// TwinCAT 3 PLC project Untitled1
// ProgramVersion: 3.1.4022.7
// libraries:
//   Tc2_Standard, * (Beckhoff Automation GmbH)
//   Tc2_System, * (Beckhoff Automation GmbH)
//   Tc3_Module, * (Beckhoff Automation GmbH)
// project tree:
//   CIF/ alg_a_DledQ1.TcPOU, alg_a_DledQ2.TcPOU, alg_a_Dresetled.TcPOU, alg_a_Dstartled.TcPOU, alg_a_ejectpulse.TcPOU, alg_a_gripperclose.TcPOU, alg_a_handlingready.TcPOU, alg_a_HledQ1.TcPOU, alg_a_HledQ2.TcPOU, alg_a_Hresetled.TcPOU, alg_a_Hstartled.TcPOU, alg_a_pusher1.TcPOU, alg_a_pusher2.TcPOU, alg_a_pusher3.TcPOU, alg_a_transfer2droppos.TcPOU, alg_a_transfer2pickpos.TcPOU, alg_a_vacuum.TcPOU, alg_a_x2distributing.TcPOU, alg_a_x2testing.TcPOU, alg_a_zdown.TcPOU, alg_M_example_controller_a_Dstartled.TcPOU, alg_M_example_controller_godown.TcPOU, alg_s_Dinitialized.TcPOU, alg_s_Hinitialized.TcPOU, derivcvar_M_HardwareMap_t.TcPOU, enum_E.TcDUT, INPUTS.TcGVL, MAIN.TcPOU, makeArray0.TcPOU, normProjIdx.TcPOU, projArray0.TcPOU, STATE.TcDUT, TIMERS.TcGVL
//   / PlcTask.TcTTO
//   UNITY/ ACTUATOR.TcPOU (not stored), GVLS.TcGVL (not stored), INDICATORLIGHT.TcPOU (not stored), UNITY.TcPOU
// real-time tasks:
//   TASK PlcTask: cycle T#10ms, priority 20, ADS port 350

CONFIGURATION Untitled1
    RESOURCE PLC ON TwinCAT3
        TASK PlcTask(INTERVAL := T#10ms, PRIORITY := 20);
        PROGRAM MAIN WITH PlcTask : MAIN;
        PROGRAM UNITY WITH PlcTask : UNITY;
    END_RESOURCE
END_CONFIGURATION

// ---- CIF/enum_E.TcDUT
TYPE enum_E :
(
	elit_gopickup,
	elit_init0,
	elit_init1,
	elit_init2,
	elit_init3,
	elit_init4,
	elit_init5,
	elit_init6,
	elit_init7,
	elit_init8,
	elit_init9,
	elit_init_error,
	elit_init_ok,
	elit_init_sensor_check,
	elit_initialized,
	elit_running,
	elit_starting,
	elit_wait_init,
	elit_wait_start
);
END_TYPE

// ---- CIF/STATE.TcDUT
TYPE STATE :
STRUCT
	curTime: LREAL;
	dvar_M_example_controller_a_x2distributing AT %Q*: BOOL;
	dvar_M_example_controller_a_zdown AT %Q*: BOOL;
	dvar_M_example_controller_count AT %Q*: DINT;
	dvar_M_example_controller AT %Q*: enum_E;
	dvar_M_HardwareMap_out_a_Dstartled AT %Q*: BOOL;
	dvar_M_HardwareMap_out_a_Dresetled AT %Q*: BOOL;
	dvar_M_HardwareMap_out_a_DledQ1 AT %Q*: BOOL;
	dvar_M_HardwareMap_out_a_DledQ2 AT %Q*: BOOL;
	dvar_M_HardwareMap_out_a_Dout4 AT %Q*: BOOL;
	dvar_M_HardwareMap_out_a_Dout5 AT %Q*: BOOL;
	dvar_M_HardwareMap_out_a_Dout6 AT %Q*: BOOL;
	dvar_M_HardwareMap_out_a_Dout7 AT %Q*: BOOL;
	dvar_M_HardwareMap_out_a_pusher1 AT %Q*: BOOL;
	dvar_M_HardwareMap_out_a_pusher2 AT %Q*: BOOL;
	dvar_M_HardwareMap_out_a_pusher3 AT %Q*: BOOL;
	dvar_M_HardwareMap_out_a_Hstartled AT %Q*: BOOL;
	dvar_M_HardwareMap_out_a_Hresetled AT %Q*: BOOL;
	dvar_M_HardwareMap_out_a_HledQ1 AT %Q*: BOOL;
	dvar_M_HardwareMap_out_a_HledQ2 AT %Q*: BOOL;
	dvar_M_HardwareMap_out_a_Hout4 AT %Q*: BOOL;
	dvar_M_HardwareMap_out_a_Hout5 AT %Q*: BOOL;
	dvar_M_HardwareMap_out_a_Hout6 AT %Q*: BOOL;
	dvar_M_HardwareMap_out_a_Hout7 AT %Q*: BOOL;
	dvar_M_HardwareMap_out_a_x2distributing AT %Q*: BOOL;
	dvar_M_HardwareMap_out_a_x2testing AT %Q*: BOOL;
	dvar_M_HardwareMap_out_a_zdown AT %Q*: BOOL;
	dvar_M_HardwareMap_out_a_gripperclose AT %Q*: BOOL;
	dvar_M_HardwareMap_out_a_transfer2pickpos AT %Q*: BOOL;
	dvar_M_HardwareMap_out_a_transfer2droppos AT %Q*: BOOL;
	dvar_M_HardwareMap_out_a_vacuum AT %Q*: BOOL;
	dvar_M_HardwareMap_out_a_ejectpulse AT %Q*: BOOL;
	dvar_M_HardwareMap_out_a_handlingready AT %Q*: BOOL;
	dvar_M_HardwareMap_init_err_sen_idx AT %Q*: DINT;
	dvar_M_HardwareMap_init_err_led_idx AT %Q*: DINT;
	cvar_M_HardwareMap_t AT %Q*: LREAL;
	dvar_M_HardwareMap AT %Q*: enum_E;
END_STRUCT
END_TYPE

// ---- CIF/INPUTS.TcGVL
VAR_GLOBAL
	ivar_s_Dstartbutton AT %I*: BOOL;
	ivar_s_Dstopbutton AT %I*: BOOL;
	ivar_s_Dresetbutton AT %I*: BOOL;
	ivar_s_Dautoswitch AT %I*: BOOL;
	ivar_s_pusher1_in AT %I*: BOOL;
	ivar_s_pusher1_out AT %I*: BOOL;
	ivar_s_stack1filled AT %I*: BOOL;
	ivar_s_product1 AT %I*: BOOL;
	ivar_s_pusher2_in AT %I*: BOOL;
	ivar_s_pusher2_out AT %I*: BOOL;
	ivar_s_stack2filled AT %I*: BOOL;
	ivar_s_product2 AT %I*: BOOL;
	ivar_s_pusher3_in AT %I*: BOOL;
	ivar_s_pusher3_out AT %I*: BOOL;
	ivar_s_stack3filled AT %I*: BOOL;
	ivar_s_product3 AT %I*: BOOL;
	ivar_s_handlingbusy AT %I*: BOOL;
	ivar_s_Hstartbutton AT %I*: BOOL;
	ivar_s_Hstopbutton AT %I*: BOOL;
	ivar_s_Hresetbutton AT %I*: BOOL;
	ivar_s_Hautoswitch AT %I*: BOOL;
	ivar_s_xpos_at1 AT %I*: BOOL;
	ivar_s_xpos_at2 AT %I*: BOOL;
	ivar_s_xpos_at3 AT %I*: BOOL;
	ivar_s_xpos_atdrop AT %I*: BOOL;
	ivar_s_zpos_atup AT %I*: BOOL;
	ivar_s_zpos_atdown AT %I*: BOOL;
	ivar_s_gripper AT %I*: BOOL;
	ivar_s_transfer_atpickup AT %I*: BOOL;
	ivar_s_transfer_atdrop AT %I*: BOOL;
	ivar_s_transfer_athalfway AT %I*: BOOL;
	ivar_s_vacuum AT %I*: BOOL;
	ivar_s_product4 AT %I*: BOOL;
	ivar_s_testingbusy AT %I*: BOOL;
	ivar_s_Din4 AT %I*: BOOL;
	ivar_s_Din5 AT %I*: BOOL;
	ivar_s_Din6 AT %I*: BOOL;
	ivar_s_Din7 AT %I*: BOOL;
	ivar_s_Hin4 AT %I*: BOOL;
	ivar_s_Hin5 AT %I*: BOOL;
	ivar_s_Hin6 AT %I*: BOOL;
	ivar_s_Hin7 AT %I*: BOOL;
	ivar_a_Dout4 AT %I*: BOOL;
	ivar_a_Dout5 AT %I*: BOOL;
	ivar_a_Dout6 AT %I*: BOOL;
	ivar_a_Dout7 AT %I*: BOOL;
	ivar_a_Hout4 AT %I*: BOOL;
	ivar_a_Hout5 AT %I*: BOOL;
	ivar_a_Hout6 AT %I*: BOOL;
	ivar_a_Hout7 AT %I*: BOOL;
END_VAR

// ---- CIF/TIMERS.TcGVL
VAR_GLOBAL
	timer0: TON;
	timer1: TON;
	curTimer: INT := 0;
END_VAR

// ---- CIF/MAIN.TcPOU
PROGRAM MAIN
VAR_OUTPUT
	timerValue0: TIME;
	timerValue1: TIME;
END_VAR
VAR
	cnt: LINT;
	first: BOOL := TRUE;
	curTimerValue: TIME;
	state0: STATE;
	curTime: LREAL;
	loopsKilled: LINT;
END_VAR
VAR_TEMP
	lastTimerValue: TIME;
	curDeltaTime: TIME;
	curDeltaSecs: LREAL;
	state1: STATE;
	progress: BOOL;
	loopCount: INT;
	b1: BOOL;
	b2: BOOL;
END_VAR


// Handle 'time' and cycle time.
cnt := cnt + 1;

timer0(IN := curTimer = 0, PT := T#1D);
timer1(IN := curTimer = 1, PT := T#1D);
timerValue0 := timer0.ET;
timerValue1 := timer1.ET;

lastTimerValue := curTimerValue;
IF curTimer = 0 THEN
    curTimerValue := timerValue0;
ELSE
    curTimerValue := timerValue1;
END_IF;
curDeltaTime := curTimerValue - lastTimerValue;
curDeltaSecs := TIME_TO_LREAL(curDeltaTime) / 1000;
curTime := curTime + curDeltaSecs;

IF cnt MOD 10 = 0 THEN
    curTimer := 1 - curTimer;
    curTimerValue := T#0S;
    timer0(IN := curTimer = 0, PT := T#1D);
    timer1(IN := curTimer = 1, PT := T#1D);
    timerValue0 := timer0.ET;
    timerValue1 := timer1.ET;
END_IF;

IF first THEN
    first := FALSE;

    // Initialize state variables for initial state.
    state0.dvar_M_example_controller_a_x2distributing := FALSE;
    state0.dvar_M_example_controller_a_zdown := FALSE;
    state0.dvar_M_example_controller_a_gripperclose := FALSE;
    state0.dvar_M_example_controller_a_x2testing := FALSE;
    state0.dvar_M_example_controller_i := 0;
    state0.cvar_M_example_controller_t := 0.0;
    state0.dvar_M_example_controller := elit_init2;
    state0.dvar_M_HardwareMap_out_a_Dstartled := FALSE;
    state0.dvar_M_HardwareMap_out_a_Dresetled := FALSE;
    state0.dvar_M_HardwareMap_out_a_DledQ1 := TRUE;
    state0.dvar_M_HardwareMap_out_a_DledQ2 := TRUE;
    state0.dvar_M_HardwareMap_out_a_Dout4 := FALSE;
    state0.dvar_M_HardwareMap_out_a_Dout5 := FALSE;
    state0.dvar_M_HardwareMap_out_a_Dout6 := FALSE;
    state0.dvar_M_HardwareMap_out_a_Dout7 := FALSE;
    state0.dvar_M_HardwareMap_out_a_pusher1 := FALSE;
    state0.dvar_M_HardwareMap_out_a_pusher2 := FALSE;
    state0.dvar_M_HardwareMap_out_a_pusher3 := FALSE;
    state0.dvar_M_HardwareMap_out_a_Hstartled := FALSE;
    state0.dvar_M_HardwareMap_out_a_Hresetled := FALSE;
    state0.dvar_M_HardwareMap_out_a_HledQ1 := TRUE;
    state0.dvar_M_HardwareMap_out_a_HledQ2 := TRUE;
    state0.dvar_M_HardwareMap_out_a_Hout4 := FALSE;
    state0.dvar_M_HardwareMap_out_a_Hout5 := FALSE;
    state0.dvar_M_HardwareMap_out_a_Hout6 := FALSE;
    state0.dvar_M_HardwareMap_out_a_Hout7 := FALSE;
    state0.dvar_M_HardwareMap_out_a_x2distributing := TRUE;
    state0.dvar_M_HardwareMap_out_a_x2testing := TRUE;
    state0.dvar_M_HardwareMap_out_a_zdown := FALSE;
    state0.dvar_M_HardwareMap_out_a_gripperclose := FALSE;
    state0.dvar_M_HardwareMap_out_a_transfer2pickpos := FALSE;
    state0.dvar_M_HardwareMap_out_a_transfer2droppos := FALSE;
    state0.dvar_M_HardwareMap_out_a_vacuum := FALSE;
    state0.dvar_M_HardwareMap_out_a_ejectpulse := FALSE;
    state0.dvar_M_HardwareMap_out_a_handlingready := FALSE;
    state0.dvar_M_HardwareMap_init_err_sen_idx := -1;
    state0.dvar_M_HardwareMap_init_err_led_idx := 0;
    state0.cvar_M_HardwareMap_t := 0.0;
    state0.dvar_M_HardwareMap := elit_init0;
    state0.dvar_M_inventory1_a_pusher1 := FALSE;
    state0.dvar_M_inventory1 := elit_init2;
    state0.dvar_M_inventory2_a_pusher2 := FALSE;
    state0.dvar_M_inventory2 := elit_init2;
    state0.dvar_M_inventory3_a_pusher3 := FALSE;
    state0.dvar_M_inventory3 := elit_init2;
    state0.dvar_M_vacuum_a_transfer2pickpos := FALSE;
    state0.dvar_M_vacuum_a_transfer2droppos := FALSE;
    state0.dvar_M_vacuum_a_vacuum := FALSE;
    state0.dvar_M_vacuum_a_ejectpulse := FALSE;
    state0.dvar_M_vacuum := elit_init2;
ELSE
    // Update continuous variables for time delay.
    state1.cvar_M_example_controller_t := state0.cvar_M_example_controller_t + curDeltaSecs * derivcvar_M_example_controller_t(state0);
    state1.cvar_M_HardwareMap_t := state0.cvar_M_HardwareMap_t + curDeltaSecs * derivcvar_M_HardwareMap_t(state0);

    state0.curTime := curTime;
    state0.cvar_M_example_controller_t := state1.cvar_M_example_controller_t;
    state0.cvar_M_HardwareMap_t := state1.cvar_M_HardwareMap_t;
END_IF;

// Event loop.
WHILE TRUE DO
    progress := FALSE;

    // Event "tau".
    IF NOT progress THEN
        b1 := (state0.dvar_M_example_controller) = (elit_init2);
        b1 := b1 AND (alg_s_Dinitialized(state0));
        IF b1 THEN
            progress := TRUE;
            state1 := state0;

            state1.dvar_M_example_controller := elit_wait_start;

            state0 := state1;
        END_IF;
    END_IF;

    // Event "tau".
    IF NOT progress THEN
        b1 := (state0.dvar_M_example_controller) = (elit_wait_start);
        b1 := b1 AND (ivar_s_Dstartbutton);
        IF b1 THEN
            progress := TRUE;
            state1 := state0;

            state1.dvar_M_example_controller := elit_droppoint;

            state0 := state1;
        END_IF;
    END_IF;

    // Event "tau".
    IF NOT progress THEN
        b1 := (state0.dvar_M_example_controller) = (elit_droppoint);
        b1 := b1 AND (ivar_s_gripper);
        b1 := b1 AND (ivar_s_xpos_atdrop);
        b1 := b1 AND (ivar_s_zpos_atup);
        IF b1 THEN
            progress := TRUE;
            state1 := state0;

            state1.dvar_M_example_controller_a_x2distributing := TRUE;
            state1.dvar_M_example_controller_a_x2testing := TRUE;
            state1.dvar_M_example_controller := elit_down;

            state0 := state1;
        END_IF;
    END_IF;

    // Event "tau".
    IF NOT progress THEN
        b1 := (state0.dvar_M_example_controller) = (elit_droppoint);
        b1 := b1 AND (NOT(ivar_s_gripper));
        b1 := b1 AND (ivar_s_xpos_atdrop);
        IF b1 THEN
            progress := TRUE;
            state1 := state0;

            state1.dvar_M_example_controller_a_x2distributing := TRUE;
            state1.dvar_M_example_controller_a_x2testing := FALSE;
            state1.dvar_M_example_controller := elit_movetopickup;

            state0 := state1;
        END_IF;
    END_IF;

    // Event "tau".
    IF NOT progress THEN
        b1 := (state0.dvar_M_example_controller) = (elit_movetopickup);
        b1 := b1 AND (projArray1(alg_M_example_controller_atpos(state0), projArray0(makeArray0(0, 1, 0, 2), state0.dvar_M_example_controller_i)));
        b1 := b1 AND ((state0.dvar_M_example_controller_i) < (3));
        IF b1 THEN
            progress := TRUE;
            state1 := state0;

            state1.dvar_M_example_controller_i := (state0.dvar_M_example_controller_i) + (1);
            state1.dvar_M_example_controller_a_x2distributing := TRUE;
            state1.dvar_M_example_controller_a_x2testing := TRUE;
            state1.dvar_M_example_controller := elit_down;

            state0 := state1;
        END_IF;
    END_IF;

    // Event "tau".
    IF NOT progress THEN
        b1 := (state0.dvar_M_example_controller) = (elit_movetopickup);
        b1 := b1 AND (projArray1(alg_M_example_controller_atpos(state0), projArray0(makeArray0(0, 1, 0, 2), state0.dvar_M_example_controller_i)));
        b1 := b1 AND ((state0.dvar_M_example_controller_i) >= (3));
        IF b1 THEN
            progress := TRUE;
            state1 := state0;

            state1.dvar_M_example_controller_i := 0;
            state1.dvar_M_example_controller_a_x2distributing := TRUE;
            state1.dvar_M_example_controller_a_x2testing := TRUE;
            state1.dvar_M_example_controller := elit_down;

            state0 := state1;
        END_IF;
    END_IF;

    // Event "tau".
    IF NOT progress THEN
        IF (state0.dvar_M_example_controller) = (elit_down) THEN
            progress := TRUE;
            state1 := state0;

            state1.dvar_M_example_controller_a_zdown := TRUE;
            state1.dvar_M_example_controller := elit_gopickup;

            state0 := state1;
        END_IF;
    END_IF;

    // Event "tau".
    IF NOT progress THEN
        b1 := (state0.dvar_M_example_controller) = (elit_gopickup);
        b1 := b1 AND (ivar_s_zpos_atdown);
        b1 := b1 AND (ivar_s_gripper);
        b1 := b1 AND (NOT(ivar_s_xpos_atdrop));
        IF b1 THEN
            progress := TRUE;
            state1 := state0;

            state1.dvar_M_example_controller_a_gripperclose := TRUE;
            state1.dvar_M_example_controller_a_zdown := FALSE;
            state1.dvar_M_example_controller := elit_goback;

            state0 := state1;
        END_IF;
    END_IF;

    // Event "tau".
    IF NOT progress THEN
        b1 := (state0.dvar_M_example_controller) = (elit_gopickup);
        b1 := b1 AND (ivar_s_zpos_atdown);
        b1 := b1 AND (ivar_s_gripper);
        b1 := b1 AND (ivar_s_xpos_atdrop);
        IF b1 THEN
            progress := TRUE;
            state1 := state0;

            state1.dvar_M_example_controller_a_gripperclose := FALSE;
            state1.dvar_M_example_controller_a_zdown := FALSE;
            state1.dvar_M_example_controller := elit_droppoint;

            state0 := state1;
        END_IF;
    END_IF;

    // Event "tau".
    IF NOT progress THEN
        b1 := (state0.dvar_M_example_controller) = (elit_gopickup);
        b1 := b1 AND (ivar_s_zpos_atdown);
        b1 := b1 AND (NOT(ivar_s_gripper));
        b1 := b1 AND (NOT(ivar_s_xpos_atdrop));
        IF b1 THEN
            progress := TRUE;
            state1 := state0;

            state1.dvar_M_example_controller_a_zdown := FALSE;
            state1.dvar_M_example_controller_a_x2distributing := FALSE;
            state1.dvar_M_example_controller_a_x2testing := TRUE;
            state1.dvar_M_example_controller := elit_finished;

            state0 := state1;
        END_IF;
    END_IF;

    // Event "tau".
    IF NOT progress THEN
        b1 := (state0.dvar_M_example_controller) = (elit_goback);
        b1 := b1 AND (ivar_s_zpos_atup);
        b1 := b1 AND (ivar_s_gripper);
        b1 := b1 AND ((state0.cvar_M_example_controller_t) > (1));
        IF b1 THEN
            progress := TRUE;
            state1 := state0;

            state1.dvar_M_example_controller_a_x2testing := TRUE;
            state1.dvar_M_example_controller_a_x2distributing := FALSE;
            state1.cvar_M_example_controller_t := 0.0;
            state1.dvar_M_example_controller := elit_droppoint;

            state0 := state1;
        END_IF;
    END_IF;

    // Event "tau".
    IF NOT progress THEN
        b1 := (state0.dvar_M_example_controller) = (elit_finished);
        b1 := b1 AND (ivar_s_xpos_atdrop);
        IF b1 THEN
            progress := TRUE;
            state1 := state0;

            state1.dvar_M_example_controller_a_x2distributing := TRUE;
            state1.dvar_M_example_controller_a_x2testing := TRUE;
            state1.dvar_M_example_controller := elit_reset;

            state0 := state1;
        END_IF;
    END_IF;

    // Event "tau".
    IF NOT progress THEN
        b1 := (state0.dvar_M_example_controller) = (elit_reset);
        b1 := b1 AND ((state0.cvar_M_example_controller_t) > (1));
        IF b1 THEN
            progress := TRUE;
            state1 := state0;

            state1.dvar_M_example_controller_a_x2distributing := FALSE;
            state1.dvar_M_example_controller_a_x2testing := FALSE;
            state1.dvar_M_example_controller := elit_wait_start;

            state0 := state1;
        END_IF;
    END_IF;

    // Event "tau".
    IF NOT progress THEN
        b1 := (state0.dvar_M_HardwareMap) = (elit_init0);
        b1 := b1 AND ((state0.cvar_M_HardwareMap_t) >= (2.0));
        IF b1 THEN
            progress := TRUE;
            state1 := state0;

            state1.dvar_M_HardwareMap := elit_init1;

            state0 := state1;
        END_IF;
    END_IF;

    // Event "tau".
    IF NOT progress THEN
        IF (state0.dvar_M_HardwareMap) = (elit_init1) THEN
            progress := TRUE;
            state1 := state0;

            state1.dvar_M_HardwareMap_out_a_x2testing := FALSE;
            state1.dvar_M_HardwareMap := elit_init2;

            state0 := state1;
        END_IF;
    END_IF;

    // Event "tau".
    IF NOT progress THEN
        b1 := (state0.dvar_M_HardwareMap) = (elit_init2);
        IF b1 THEN
            b2 := ivar_s_xpos_at1;
            b2 := b2 OR (ivar_s_xpos_at2);
            b1 := b1 AND (b2);
        END_IF;
        IF b1 THEN
            progress := TRUE;
            state1 := state0;

            state1.dvar_M_HardwareMap_out_a_x2testing := TRUE;
            state1.dvar_M_HardwareMap := elit_init3;

            state0 := state1;
        END_IF;
    END_IF;

    // Event "tau".
    IF NOT progress THEN
        IF (state0.dvar_M_HardwareMap) = (elit_init3) THEN
            progress := TRUE;
            state1 := state0;

            state1.dvar_M_HardwareMap_out_a_transfer2pickpos := TRUE;
            state1.dvar_M_HardwareMap := elit_init4;

            state0 := state1;
        END_IF;
    END_IF;

    // Event "tau".
    IF NOT progress THEN
        b1 := (state0.dvar_M_HardwareMap) = (elit_init4);
        b1 := b1 AND (ivar_s_transfer_atpickup);
        IF b1 THEN
            progress := TRUE;
            state1 := state0;

            state1.dvar_M_HardwareMap_out_a_transfer2pickpos := FALSE;
            state1.dvar_M_HardwareMap := elit_init5;

            state0 := state1;
        END_IF;
    END_IF;

    // Event "tau".
    IF NOT progress THEN
        IF (state0.dvar_M_HardwareMap) = (elit_init5) THEN
            progress := TRUE;
            state1 := state0;

            state1.dvar_M_HardwareMap_out_a_transfer2droppos := TRUE;
            state1.dvar_M_HardwareMap := elit_init6;

            state0 := state1;
        END_IF;
    END_IF;

    // Event "tau".
    IF NOT progress THEN
        b1 := (state0.dvar_M_HardwareMap) = (elit_init6);
        b1 := b1 AND (ivar_s_transfer_athalfway);
        IF b1 THEN
            progress := TRUE;
            state1 := state0;

            state1.dvar_M_HardwareMap_out_a_transfer2droppos := FALSE;
            state1.dvar_M_HardwareMap := elit_init7;

            state0 := state1;
        END_IF;
    END_IF;

    // Event "tau".
    IF NOT progress THEN
        IF (state0.dvar_M_HardwareMap) = (elit_init7) THEN
            progress := TRUE;
            state1 := state0;

            state1.dvar_M_HardwareMap_out_a_x2distributing := FALSE;
            state1.dvar_M_HardwareMap := elit_init8;

            state0 := state1;
        END_IF;
    END_IF;

    // Event "tau".
    IF NOT progress THEN
        b1 := (state0.dvar_M_HardwareMap) = (elit_init8);
        b1 := b1 AND (ivar_s_xpos_atdrop);
        IF b1 THEN
            progress := TRUE;
            state1 := state0;

            state1.dvar_M_HardwareMap_out_a_x2distributing := TRUE;
            state1.cvar_M_HardwareMap_t := 0.0;
            state1.dvar_M_HardwareMap := elit_init9;

            state0 := state1;
        END_IF;
    END_IF;

    // Event "tau".
    IF NOT progress THEN
        b1 := (state0.dvar_M_HardwareMap) = (elit_init9);
        b1 := b1 AND ((state0.cvar_M_HardwareMap_t) >= (1));
        IF b1 THEN
            progress := TRUE;
            state1 := state0;

            state1.dvar_M_HardwareMap := elit_init_sensor_check;

            state0 := state1;
        END_IF;
    END_IF;

    // Event "tau".
    IF NOT progress THEN
        b1 := (state0.dvar_M_HardwareMap) = (elit_init_sensor_check);
        b1 := b1 AND (ivar_s_Dstartbutton);
        IF b1 THEN
            progress := TRUE;
            state1 := state0;

            state1.dvar_M_HardwareMap_init_err_sen_idx := 0;
            state1.dvar_M_HardwareMap := elit_init_error;

            state0 := state1;
        END_IF;
    END_IF;

    // Event "tau".
    IF NOT progress THEN
        b1 := (state0.dvar_M_HardwareMap) = (elit_init_sensor_check);
        b1 := b1 AND (NOT(ivar_s_Dstopbutton));
        IF b1 THEN
            progress := TRUE;
            state1 := state0;

            state1.dvar_M_HardwareMap_init_err_sen_idx := 1;
            state1.dvar_M_HardwareMap := elit_init_error;

            state0 := state1;
        END_IF;
    END_IF;

    // Event "tau".
    IF NOT progress THEN
        b1 := (state0.dvar_M_HardwareMap) = (elit_init_sensor_check);
        b1 := b1 AND (ivar_s_Dautoswitch);
        IF b1 THEN
            progress := TRUE;
            state1 := state0;

            state1.dvar_M_HardwareMap_init_err_sen_idx := 2;
            state1.dvar_M_HardwareMap := elit_init_error;

            state0 := state1;
        END_IF;
    END_IF;

    // Event "tau".
    IF NOT progress THEN
        b1 := (state0.dvar_M_HardwareMap) = (elit_init_sensor_check);
        b1 := b1 AND (ivar_s_Dresetbutton);
        IF b1 THEN
            progress := TRUE;
            state1 := state0;

            state1.dvar_M_HardwareMap_init_err_sen_idx := 3;
            state1.dvar_M_HardwareMap := elit_init_error;

            state0 := state1;
        END_IF;
    END_IF;

    // Event "tau".
    IF NOT progress THEN
        b1 := (state0.dvar_M_HardwareMap) = (elit_init_sensor_check);
        b1 := b1 AND (ivar_s_Din4);
        IF b1 THEN
            progress := TRUE;
            state1 := state0;

            state1.dvar_M_HardwareMap_init_err_sen_idx := 4;
            state1.dvar_M_HardwareMap := elit_init_error;

            state0 := state1;
        END_IF;
    END_IF;

    // Event "tau".
    IF NOT progress THEN
        b1 := (state0.dvar_M_HardwareMap) = (elit_init_sensor_check);
        b1 := b1 AND (ivar_s_Din5);
        IF b1 THEN
            progress := TRUE;
            state1 := state0;

            state1.dvar_M_HardwareMap_init_err_sen_idx := 5;
            state1.dvar_M_HardwareMap := elit_init_error;

            state0 := state1;
        END_IF;
    END_IF;

    // Event "tau".
    IF NOT progress THEN
        b1 := (state0.dvar_M_HardwareMap) = (elit_init_sensor_check);
        b1 := b1 AND (ivar_s_Din6);
        IF b1 THEN
            progress := TRUE;
            state1 := state0;

            state1.dvar_M_HardwareMap_init_err_sen_idx := 6;
            state1.dvar_M_HardwareMap := elit_init_error;

            state0 := state1;
        END_IF;
    END_IF;

    // Event "tau".
    IF NOT progress THEN
        b1 := (state0.dvar_M_HardwareMap) = (elit_init_sensor_check);
        b1 := b1 AND (ivar_s_Din7);
        IF b1 THEN
            progress := TRUE;
            state1 := state0;

            state1.dvar_M_HardwareMap_init_err_sen_idx := 7;
            state1.dvar_M_HardwareMap := elit_init_error;

            state0 := state1;
        END_IF;
    END_IF;

    // Event "tau".
    IF NOT progress THEN
        b1 := (state0.dvar_M_HardwareMap) = (elit_init_sensor_check);
        b1 := b1 AND (NOT(ivar_s_pusher1_in));
        IF b1 THEN
            progress := TRUE;
            state1 := state0;

            state1.dvar_M_HardwareMap_init_err_sen_idx := 8;
            state1.dvar_M_HardwareMap := elit_init_error;

            state0 := state1;
        END_IF;
    END_IF;

    // Event "tau".
    IF NOT progress THEN
        b1 := (state0.dvar_M_HardwareMap) = (elit_init_sensor_check);
        b1 := b1 AND (ivar_s_pusher1_out);
        IF b1 THEN
            progress := TRUE;
            state1 := state0;

            state1.dvar_M_HardwareMap_init_err_sen_idx := 9;
            state1.dvar_M_HardwareMap := elit_init_error;

            state0 := state1;
        END_IF;
    END_IF;

    // Event "tau".
    IF NOT progress THEN
        b1 := (state0.dvar_M_HardwareMap) = (elit_init_sensor_check);
        b1 := b1 AND (NOT(ivar_s_stack1filled));
        IF b1 THEN
            progress := TRUE;
            state1 := state0;

            state1.dvar_M_HardwareMap_init_err_sen_idx := 10;
            state1.dvar_M_HardwareMap := elit_init_error;

            state0 := state1;
        END_IF;
    END_IF;

    // Event "tau".
    IF NOT progress THEN
        b1 := (state0.dvar_M_HardwareMap) = (elit_init_sensor_check);
        b1 := b1 AND (ivar_s_product1);
        IF b1 THEN
            progress := TRUE;
            state1 := state0;

            state1.dvar_M_HardwareMap_init_err_sen_idx := 11;
            state1.dvar_M_HardwareMap := elit_init_error;

            state0 := state1;
        END_IF;
    END_IF;

    // Event "tau".
    IF NOT progress THEN
        b1 := (state0.dvar_M_HardwareMap) = (elit_init_sensor_check);
        b1 := b1 AND (NOT(ivar_s_pusher2_in));
        IF b1 THEN
            progress := TRUE;
            state1 := state0;

            state1.dvar_M_HardwareMap_init_err_sen_idx := 12;
            state1.dvar_M_HardwareMap := elit_init_error;

            state0 := state1;
        END_IF;
    END_IF;

    // Event "tau".
    IF NOT progress THEN
        b1 := (state0.dvar_M_HardwareMap) = (elit_init_sensor_check);
        b1 := b1 AND (ivar_s_pusher2_out);
        IF b1 THEN
            progress := TRUE;
            state1 := state0;

            state1.dvar_M_HardwareMap_init_err_sen_idx := 13;
            state1.dvar_M_HardwareMap := elit_init_error;

            state0 := state1;
        END_IF;
    END_IF;

    // Event "tau".
    IF NOT progress THEN
        b1 := (state0.dvar_M_HardwareMap) = (elit_init_sensor_check);
        b1 := b1 AND (NOT(ivar_s_stack2filled));
        IF b1 THEN
            progress := TRUE;
            state1 := state0;

            state1.dvar_M_HardwareMap_init_err_sen_idx := 14;
            state1.dvar_M_HardwareMap := elit_init_error;

            state0 := state1;
        END_IF;
    END_IF;

    // Event "tau".
    IF NOT progress THEN
        b1 := (state0.dvar_M_HardwareMap) = (elit_init_sensor_check);
        b1 := b1 AND (ivar_s_product2);
        IF b1 THEN
            progress := TRUE;
            state1 := state0;

            state1.dvar_M_HardwareMap_init_err_sen_idx := 15;
            state1.dvar_M_HardwareMap := elit_init_error;

            state0 := state1;
        END_IF;
    END_IF;

    // Event "tau".
    IF NOT progress THEN
        b1 := (state0.dvar_M_HardwareMap) = (elit_init_sensor_check);
        b1 := b1 AND (NOT(ivar_s_pusher3_in));
        IF b1 THEN
            progress := TRUE;
            state1 := state0;

            state1.dvar_M_HardwareMap_init_err_sen_idx := 16;
            state1.dvar_M_HardwareMap := elit_init_error;

            state0 := state1;
        END_IF;
    END_IF;

    // Event "tau".
    IF NOT progress THEN
        b1 := (state0.dvar_M_HardwareMap) = (elit_init_sensor_check);
        b1 := b1 AND (ivar_s_pusher3_out);
        IF b1 THEN
            progress := TRUE;
            state1 := state0;

            state1.dvar_M_HardwareMap_init_err_sen_idx := 17;
            state1.dvar_M_HardwareMap := elit_init_error;

            state0 := state1;
        END_IF;
    END_IF;

    // Event "tau".
    IF NOT progress THEN
        b1 := (state0.dvar_M_HardwareMap) = (elit_init_sensor_check);
        b1 := b1 AND (NOT(ivar_s_stack3filled));
        IF b1 THEN
            progress := TRUE;
            state1 := state0;

            state1.dvar_M_HardwareMap_init_err_sen_idx := 18;
            state1.dvar_M_HardwareMap := elit_init_error;

            state0 := state1;
        END_IF;
    END_IF;

    // Event "tau".
    IF NOT progress THEN
        b1 := (state0.dvar_M_HardwareMap) = (elit_init_sensor_check);
        b1 := b1 AND (ivar_s_product3);
        IF b1 THEN
            progress := TRUE;
            state1 := state0;

            state1.dvar_M_HardwareMap_init_err_sen_idx := 19;
            state1.dvar_M_HardwareMap := elit_init_error;

            state0 := state1;
        END_IF;
    END_IF;

    // Event "tau".
    IF NOT progress THEN
        b1 := (state0.dvar_M_HardwareMap) = (elit_init_sensor_check);
        b1 := b1 AND (ivar_s_Hstartbutton);
        IF b1 THEN
            progress := TRUE;
            state1 := state0;

            state1.dvar_M_HardwareMap_init_err_sen_idx := 22;
            state1.dvar_M_HardwareMap := elit_init_error;

            state0 := state1;
        END_IF;
    END_IF;

    // Event "tau".
    IF NOT progress THEN
        b1 := (state0.dvar_M_HardwareMap) = (elit_init_sensor_check);
        b1 := b1 AND (NOT(ivar_s_Hstopbutton));
        IF b1 THEN
            progress := TRUE;
            state1 := state0;

            state1.dvar_M_HardwareMap_init_err_sen_idx := 23;
            state1.dvar_M_HardwareMap := elit_init_error;

            state0 := state1;
        END_IF;
    END_IF;

    // Event "tau".
    IF NOT progress THEN
        b1 := (state0.dvar_M_HardwareMap) = (elit_init_sensor_check);
        b1 := b1 AND (ivar_s_Hautoswitch);
        IF b1 THEN
            progress := TRUE;
            state1 := state0;

            state1.dvar_M_HardwareMap_init_err_sen_idx := 24;
            state1.dvar_M_HardwareMap := elit_init_error;

            state0 := state1;
        END_IF;
    END_IF;

    // Event "tau".
    IF NOT progress THEN
        b1 := (state0.dvar_M_HardwareMap) = (elit_init_sensor_check);
        b1 := b1 AND (ivar_s_Hresetbutton);
        IF b1 THEN
            progress := TRUE;
            state1 := state0;

            state1.dvar_M_HardwareMap_init_err_sen_idx := 25;
            state1.dvar_M_HardwareMap := elit_init_error;

            state0 := state1;
        END_IF;
    END_IF;

    // Event "tau".
    IF NOT progress THEN
        b1 := (state0.dvar_M_HardwareMap) = (elit_init_sensor_check);
        b1 := b1 AND (ivar_s_Hin4);
        IF b1 THEN
            progress := TRUE;
            state1 := state0;

            state1.dvar_M_HardwareMap_init_err_sen_idx := 26;
            state1.dvar_M_HardwareMap := elit_init_error;

            state0 := state1;
        END_IF;
    END_IF;

    // Event "tau".
    IF NOT progress THEN
        b1 := (state0.dvar_M_HardwareMap) = (elit_init_sensor_check);
        b1 := b1 AND (ivar_s_Hin5);
        IF b1 THEN
            progress := TRUE;
            state1 := state0;

            state1.dvar_M_HardwareMap_init_err_sen_idx := 27;
            state1.dvar_M_HardwareMap := elit_init_error;

            state0 := state1;
        END_IF;
    END_IF;

    // Event "tau".
    IF NOT progress THEN
        b1 := (state0.dvar_M_HardwareMap) = (elit_init_sensor_check);
        b1 := b1 AND (ivar_s_Hin6);
        IF b1 THEN
            progress := TRUE;
            state1 := state0;

            state1.dvar_M_HardwareMap_init_err_sen_idx := 28;
            state1.dvar_M_HardwareMap := elit_init_error;

            state0 := state1;
        END_IF;
    END_IF;

    // Event "tau".
    IF NOT progress THEN
        b1 := (state0.dvar_M_HardwareMap) = (elit_init_sensor_check);
        b1 := b1 AND (ivar_s_Hin7);
        IF b1 THEN
            progress := TRUE;
            state1 := state0;

            state1.dvar_M_HardwareMap_init_err_sen_idx := 29;
            state1.dvar_M_HardwareMap := elit_init_error;

            state0 := state1;
        END_IF;
    END_IF;

    // Event "tau".
    IF NOT progress THEN
        b1 := (state0.dvar_M_HardwareMap) = (elit_init_sensor_check);
        b1 := b1 AND (ivar_s_xpos_at1);
        IF b1 THEN
            progress := TRUE;
            state1 := state0;

            state1.dvar_M_HardwareMap_init_err_sen_idx := 33;
            state1.dvar_M_HardwareMap := elit_init_error;

            state0 := state1;
        END_IF;
    END_IF;

    // Event "tau".
    IF NOT progress THEN
        b1 := (state0.dvar_M_HardwareMap) = (elit_init_sensor_check);
        b1 := b1 AND (ivar_s_xpos_at2);
        IF b1 THEN
            progress := TRUE;
            state1 := state0;

            state1.dvar_M_HardwareMap_init_err_sen_idx := 34;
            state1.dvar_M_HardwareMap := elit_init_error;

            state0 := state1;
        END_IF;
    END_IF;

    // Event "tau".
    IF NOT progress THEN
        b1 := (state0.dvar_M_HardwareMap) = (elit_init_sensor_check);
        b1 := b1 AND (ivar_s_xpos_at3);
        IF b1 THEN
            progress := TRUE;
            state1 := state0;

            state1.dvar_M_HardwareMap_init_err_sen_idx := 35;
            state1.dvar_M_HardwareMap := elit_init_error;

            state0 := state1;
        END_IF;
    END_IF;

    // Event "tau".
    IF NOT progress THEN
        b1 := (state0.dvar_M_HardwareMap) = (elit_init_sensor_check);
        b1 := b1 AND (NOT(ivar_s_xpos_atdrop));
        IF b1 THEN
            progress := TRUE;
            state1 := state0;

            state1.dvar_M_HardwareMap_init_err_sen_idx := 36;
            state1.dvar_M_HardwareMap := elit_init_error;

            state0 := state1;
        END_IF;
    END_IF;

    // Event "tau".
    IF NOT progress THEN
        b1 := (state0.dvar_M_HardwareMap) = (elit_init_sensor_check);
        b1 := b1 AND (NOT(ivar_s_zpos_atup));
        IF b1 THEN
            progress := TRUE;
            state1 := state0;

            state1.dvar_M_HardwareMap_init_err_sen_idx := 37;
            state1.dvar_M_HardwareMap := elit_init_error;

            state0 := state1;
        END_IF;
    END_IF;

    // Event "tau".
    IF NOT progress THEN
        b1 := (state0.dvar_M_HardwareMap) = (elit_init_sensor_check);
        b1 := b1 AND (ivar_s_zpos_atdown);
        IF b1 THEN
            progress := TRUE;
            state1 := state0;

            state1.dvar_M_HardwareMap_init_err_sen_idx := 38;
            state1.dvar_M_HardwareMap := elit_init_error;

            state0 := state1;
        END_IF;
    END_IF;

    // Event "tau".
    IF NOT progress THEN
        b1 := (state0.dvar_M_HardwareMap) = (elit_init_sensor_check);
        b1 := b1 AND (ivar_s_gripper);
        IF b1 THEN
            progress := TRUE;
            state1 := state0;

            state1.dvar_M_HardwareMap_init_err_sen_idx := 39;
            state1.dvar_M_HardwareMap := elit_init_error;

            state0 := state1;
        END_IF;
    END_IF;

    // Event "tau".
    IF NOT progress THEN
        b1 := (state0.dvar_M_HardwareMap) = (elit_init_sensor_check);
        b1 := b1 AND (ivar_s_transfer_atpickup);
        IF b1 THEN
            progress := TRUE;
            state1 := state0;

            state1.dvar_M_HardwareMap_init_err_sen_idx := 40;
            state1.dvar_M_HardwareMap := elit_init_error;

            state0 := state1;
        END_IF;
    END_IF;

    // Event "tau".
    IF NOT progress THEN
        b1 := (state0.dvar_M_HardwareMap) = (elit_init_sensor_check);
        b1 := b1 AND (ivar_s_transfer_atdrop);
        IF b1 THEN
            progress := TRUE;
            state1 := state0;

            state1.dvar_M_HardwareMap_init_err_sen_idx := 41;
            state1.dvar_M_HardwareMap := elit_init_error;

            state0 := state1;
        END_IF;
    END_IF;

    // Event "tau".
    IF NOT progress THEN
        b1 := (state0.dvar_M_HardwareMap) = (elit_init_sensor_check);
        b1 := b1 AND (NOT(ivar_s_transfer_athalfway));
        IF b1 THEN
            progress := TRUE;
            state1 := state0;

            state1.dvar_M_HardwareMap_init_err_sen_idx := 42;
            state1.dvar_M_HardwareMap := elit_init_error;

            state0 := state1;
        END_IF;
    END_IF;

    // Event "tau".
    IF NOT progress THEN
        b1 := (state0.dvar_M_HardwareMap) = (elit_init_sensor_check);
        b1 := b1 AND (ivar_s_vacuum);
        IF b1 THEN
            progress := TRUE;
            state1 := state0;

            state1.dvar_M_HardwareMap_init_err_sen_idx := 43;
            state1.dvar_M_HardwareMap := elit_init_error;

            state0 := state1;
        END_IF;
    END_IF;

    // Event "tau".
    IF NOT progress THEN
        b1 := (state0.dvar_M_HardwareMap) = (elit_init_sensor_check);
        b1 := b1 AND (ivar_s_product4);
        IF b1 THEN
            progress := TRUE;
            state1 := state0;

            state1.dvar_M_HardwareMap_init_err_sen_idx := 44;
            state1.dvar_M_HardwareMap := elit_init_error;

            state0 := state1;
        END_IF;
    END_IF;

    // Event "tau".
    IF NOT progress THEN
        b1 := (state0.dvar_M_HardwareMap) = (elit_init_sensor_check);
        b1 := b1 AND (NOT(ivar_s_Dstartbutton));
        b1 := b1 AND (ivar_s_Dstopbutton);
        b1 := b1 AND (NOT(ivar_s_Dautoswitch));
        b1 := b1 AND (NOT(ivar_s_Dresetbutton));
        b1 := b1 AND (NOT(ivar_s_Din4));
        b1 := b1 AND (NOT(ivar_s_Din5));
        b1 := b1 AND (NOT(ivar_s_Din6));
        b1 := b1 AND (NOT(ivar_s_Din7));
        b1 := b1 AND (ivar_s_pusher1_in);
        b1 := b1 AND (NOT(ivar_s_pusher1_out));
        b1 := b1 AND (ivar_s_stack1filled);
        b1 := b1 AND (NOT(ivar_s_product1));
        b1 := b1 AND (ivar_s_pusher2_in);
        b1 := b1 AND (NOT(ivar_s_pusher2_out));
        b1 := b1 AND (ivar_s_stack2filled);
        b1 := b1 AND (NOT(ivar_s_product2));
        b1 := b1 AND (ivar_s_pusher3_in);
        b1 := b1 AND (NOT(ivar_s_pusher3_out));
        b1 := b1 AND (ivar_s_stack3filled);
        b1 := b1 AND (NOT(ivar_s_product3));
        b1 := b1 AND (NOT(ivar_s_Hstartbutton));
        b1 := b1 AND (ivar_s_Hstopbutton);
        b1 := b1 AND (NOT(ivar_s_Hautoswitch));
        b1 := b1 AND (NOT(ivar_s_Hresetbutton));
        b1 := b1 AND (NOT(ivar_s_Hin4));
        b1 := b1 AND (NOT(ivar_s_Hin5));
        b1 := b1 AND (NOT(ivar_s_Hin6));
        b1 := b1 AND (NOT(ivar_s_Hin7));
        b1 := b1 AND (NOT(ivar_s_xpos_at1));
        b1 := b1 AND (NOT(ivar_s_xpos_at2));
        b1 := b1 AND (NOT(ivar_s_xpos_at3));
        b1 := b1 AND (ivar_s_xpos_atdrop);
        b1 := b1 AND (ivar_s_zpos_atup);
        b1 := b1 AND (NOT(ivar_s_zpos_atdown));
        b1 := b1 AND (NOT(ivar_s_gripper));
        b1 := b1 AND (NOT(ivar_s_transfer_atpickup));
        b1 := b1 AND (NOT(ivar_s_transfer_atdrop));
        b1 := b1 AND (ivar_s_transfer_athalfway);
        b1 := b1 AND (NOT(ivar_s_vacuum));
        b1 := b1 AND (NOT(ivar_s_product4));
        IF b1 THEN
            progress := TRUE;
            state1 := state0;

            state1.dvar_M_HardwareMap := elit_init_ok;

            state0 := state1;
        END_IF;
    END_IF;

    // Event "tau".
    IF NOT progress THEN
        b1 := (state0.dvar_M_HardwareMap) = (elit_init_error);
        b1 := b1 AND ((state0.cvar_M_HardwareMap_t) >= (0.5));
        b1 := b1 AND ((state0.dvar_M_HardwareMap_init_err_led_idx) = (0));
        IF b1 THEN
            progress := TRUE;
            state1 := state0;

            state1.cvar_M_HardwareMap_t := 0.0;
            state1.dvar_M_HardwareMap_init_err_led_idx := 1;
            state1.dvar_M_HardwareMap_out_a_DledQ1 := TRUE;
            state1.dvar_M_HardwareMap_out_a_DledQ2 := FALSE;
            state1.dvar_M_HardwareMap_out_a_HledQ1 := TRUE;
            state1.dvar_M_HardwareMap_out_a_HledQ2 := FALSE;

            state0 := state1;
        END_IF;
    END_IF;

    // Event "tau".
    IF NOT progress THEN
        b1 := (state0.dvar_M_HardwareMap) = (elit_init_error);
        b1 := b1 AND ((state0.cvar_M_HardwareMap_t) >= (0.5));
        b1 := b1 AND ((state0.dvar_M_HardwareMap_init_err_led_idx) = (1));
        IF b1 THEN
            progress := TRUE;
            state1 := state0;

            state1.cvar_M_HardwareMap_t := 0.0;
            state1.dvar_M_HardwareMap_init_err_led_idx := 0;
            state1.dvar_M_HardwareMap_out_a_DledQ1 := FALSE;
            state1.dvar_M_HardwareMap_out_a_DledQ2 := TRUE;
            state1.dvar_M_HardwareMap_out_a_HledQ1 := FALSE;
            state1.dvar_M_HardwareMap_out_a_HledQ2 := TRUE;

            state0 := state1;
        END_IF;
    END_IF;

    // Event "tau".
    IF NOT progress THEN
        IF (state0.dvar_M_HardwareMap) = (elit_init_ok) THEN
            progress := TRUE;
            state1 := state0;

            state1.dvar_M_HardwareMap_out_a_DledQ1 := FALSE;
            state1.dvar_M_HardwareMap_out_a_DledQ2 := FALSE;
            state1.dvar_M_HardwareMap_out_a_HledQ1 := FALSE;
            state1.dvar_M_HardwareMap_out_a_HledQ2 := FALSE;
            state1.dvar_M_HardwareMap := elit_initialized;

            state0 := state1;
        END_IF;
    END_IF;

    // Event "tau".
    IF NOT progress THEN
        b1 := (state0.dvar_M_HardwareMap) = (elit_initialized);
        b1 := b1 AND ((state0.dvar_M_HardwareMap_out_a_Dstartled) <> (alg_a_Dstartled(state0)));
        IF b1 THEN
            progress := TRUE;
            state1 := state0;

            state1.dvar_M_HardwareMap_out_a_Dstartled := alg_a_Dstartled(state0);

            state0 := state1;
        END_IF;
    END_IF;

    // Event "tau".
    IF NOT progress THEN
        b1 := (state0.dvar_M_HardwareMap) = (elit_initialized);
        b1 := b1 AND ((state0.dvar_M_HardwareMap_out_a_Dresetled) <> (FALSE));
        IF b1 THEN
            progress := TRUE;
            state1 := state0;

            state1.dvar_M_HardwareMap_out_a_Dresetled := FALSE;

            state0 := state1;
        END_IF;
    END_IF;

    // Event "tau".
    IF NOT progress THEN
        b1 := (state0.dvar_M_HardwareMap) = (elit_initialized);
        b1 := b1 AND ((state0.dvar_M_HardwareMap_out_a_DledQ1) <> (FALSE));
        IF b1 THEN
            progress := TRUE;
            state1 := state0;

            state1.dvar_M_HardwareMap_out_a_DledQ1 := FALSE;

            state0 := state1;
        END_IF;
    END_IF;

    // Event "tau".
    IF NOT progress THEN
        b1 := (state0.dvar_M_HardwareMap) = (elit_initialized);
        b1 := b1 AND ((state0.dvar_M_HardwareMap_out_a_DledQ2) <> (FALSE));
        IF b1 THEN
            progress := TRUE;
            state1 := state0;

            state1.dvar_M_HardwareMap_out_a_DledQ2 := FALSE;

            state0 := state1;
        END_IF;
    END_IF;

    // Event "tau".
    IF NOT progress THEN
        b1 := (state0.dvar_M_HardwareMap) = (elit_initialized);
        b1 := b1 AND ((state0.dvar_M_HardwareMap_out_a_Dout4) <> (ivar_a_Dout4));
        IF b1 THEN
            progress := TRUE;
            state1 := state0;

            state1.dvar_M_HardwareMap_out_a_Dout4 := ivar_a_Dout4;

            state0 := state1;
        END_IF;
    END_IF;

    // Event "tau".
    IF NOT progress THEN
        b1 := (state0.dvar_M_HardwareMap) = (elit_initialized);
        b1 := b1 AND ((state0.dvar_M_HardwareMap_out_a_Dout5) <> (ivar_a_Dout5));
        IF b1 THEN
            progress := TRUE;
            state1 := state0;

            state1.dvar_M_HardwareMap_out_a_Dout5 := ivar_a_Dout5;

            state0 := state1;
        END_IF;
    END_IF;

    // Event "tau".
    IF NOT progress THEN
        b1 := (state0.dvar_M_HardwareMap) = (elit_initialized);
        b1 := b1 AND ((state0.dvar_M_HardwareMap_out_a_Dout6) <> (ivar_a_Dout6));
        IF b1 THEN
            progress := TRUE;
            state1 := state0;

            state1.dvar_M_HardwareMap_out_a_Dout6 := ivar_a_Dout6;

            state0 := state1;
        END_IF;
    END_IF;

    // Event "tau".
    IF NOT progress THEN
        b1 := (state0.dvar_M_HardwareMap) = (elit_initialized);
        b1 := b1 AND ((state0.dvar_M_HardwareMap_out_a_Dout7) <> (ivar_a_Dout7));
        IF b1 THEN
            progress := TRUE;
            state1 := state0;

            state1.dvar_M_HardwareMap_out_a_Dout7 := ivar_a_Dout7;

            state0 := state1;
        END_IF;
    END_IF;

    // Event "tau".
    IF NOT progress THEN
        b1 := (state0.dvar_M_HardwareMap) = (elit_initialized);
        b1 := b1 AND ((state0.dvar_M_HardwareMap_out_a_pusher1) <> (alg_a_pusher1(state0)));
        IF b1 THEN
            progress := TRUE;
            state1 := state0;

            state1.dvar_M_HardwareMap_out_a_pusher1 := alg_a_pusher1(state0);

            state0 := state1;
        END_IF;
    END_IF;

    // Event "tau".
    IF NOT progress THEN
        b1 := (state0.dvar_M_HardwareMap) = (elit_initialized);
        b1 := b1 AND ((state0.dvar_M_HardwareMap_out_a_pusher2) <> (alg_a_pusher2(state0)));
        IF b1 THEN
            progress := TRUE;
            state1 := state0;

            state1.dvar_M_HardwareMap_out_a_pusher2 := alg_a_pusher2(state0);

            state0 := state1;
        END_IF;
    END_IF;

    // Event "tau".
    IF NOT progress THEN
        b1 := (state0.dvar_M_HardwareMap) = (elit_initialized);
        b1 := b1 AND ((state0.dvar_M_HardwareMap_out_a_pusher3) <> (alg_a_pusher3(state0)));
        IF b1 THEN
            progress := TRUE;
            state1 := state0;

            state1.dvar_M_HardwareMap_out_a_pusher3 := alg_a_pusher3(state0);

            state0 := state1;
        END_IF;
    END_IF;

    // Event "tau".
    IF NOT progress THEN
        b1 := (state0.dvar_M_HardwareMap) = (elit_initialized);
        b1 := b1 AND ((state0.dvar_M_HardwareMap_out_a_Hstartled) <> (FALSE));
        IF b1 THEN
            progress := TRUE;
            state1 := state0;

            state1.dvar_M_HardwareMap_out_a_Hstartled := FALSE;

            state0 := state1;
        END_IF;
    END_IF;

    // Event "tau".
    IF NOT progress THEN
        b1 := (state0.dvar_M_HardwareMap) = (elit_initialized);
        b1 := b1 AND ((state0.dvar_M_HardwareMap_out_a_Hresetled) <> (FALSE));
        IF b1 THEN
            progress := TRUE;
            state1 := state0;

            state1.dvar_M_HardwareMap_out_a_Hresetled := FALSE;

            state0 := state1;
        END_IF;
    END_IF;

    // Event "tau".
    IF NOT progress THEN
        b1 := (state0.dvar_M_HardwareMap) = (elit_initialized);
        b1 := b1 AND ((state0.dvar_M_HardwareMap_out_a_HledQ1) <> (FALSE));
        IF b1 THEN
            progress := TRUE;
            state1 := state0;

            state1.dvar_M_HardwareMap_out_a_HledQ1 := FALSE;

            state0 := state1;
        END_IF;
    END_IF;

    // Event "tau".
    IF NOT progress THEN
        b1 := (state0.dvar_M_HardwareMap) = (elit_initialized);
        b1 := b1 AND ((state0.dvar_M_HardwareMap_out_a_HledQ2) <> (FALSE));
        IF b1 THEN
            progress := TRUE;
            state1 := state0;

            state1.dvar_M_HardwareMap_out_a_HledQ2 := FALSE;

            state0 := state1;
        END_IF;
    END_IF;

    // Event "tau".
    IF NOT progress THEN
        b1 := (state0.dvar_M_HardwareMap) = (elit_initialized);
        b1 := b1 AND ((state0.dvar_M_HardwareMap_out_a_Hout4) <> (ivar_a_Hout4));
        IF b1 THEN
            progress := TRUE;
            state1 := state0;

            state1.dvar_M_HardwareMap_out_a_Hout4 := ivar_a_Hout4;

            state0 := state1;
        END_IF;
    END_IF;

    // Event "tau".
    IF NOT progress THEN
        b1 := (state0.dvar_M_HardwareMap) = (elit_initialized);
        b1 := b1 AND ((state0.dvar_M_HardwareMap_out_a_Hout5) <> (ivar_a_Hout5));
        IF b1 THEN
            progress := TRUE;
            state1 := state0;

            state1.dvar_M_HardwareMap_out_a_Hout5 := ivar_a_Hout5;

            state0 := state1;
        END_IF;
    END_IF;

    // Event "tau".
    IF NOT progress THEN
        b1 := (state0.dvar_M_HardwareMap) = (elit_initialized);
        b1 := b1 AND ((state0.dvar_M_HardwareMap_out_a_Hout6) <> (ivar_a_Hout6));
        IF b1 THEN
            progress := TRUE;
            state1 := state0;

            state1.dvar_M_HardwareMap_out_a_Hout6 := ivar_a_Hout6;

            state0 := state1;
        END_IF;
    END_IF;

    // Event "tau".
    IF NOT progress THEN
        b1 := (state0.dvar_M_HardwareMap) = (elit_initialized);
        b1 := b1 AND ((state0.dvar_M_HardwareMap_out_a_Hout7) <> (ivar_a_Hout7));
        IF b1 THEN
            progress := TRUE;
            state1 := state0;

            state1.dvar_M_HardwareMap_out_a_Hout7 := ivar_a_Hout7;

            state0 := state1;
        END_IF;
    END_IF;

    // Event "tau".
    IF NOT progress THEN
        b1 := (state0.dvar_M_HardwareMap) = (elit_initialized);
        b1 := b1 AND ((state0.dvar_M_HardwareMap_out_a_x2distributing) <> (alg_a_x2distributing(state0)));
        IF b1 THEN
            progress := TRUE;
            state1 := state0;

            state1.dvar_M_HardwareMap_out_a_x2distributing := alg_a_x2distributing(state0);

            state0 := state1;
        END_IF;
    END_IF;

    // Event "tau".
    IF NOT progress THEN
        b1 := (state0.dvar_M_HardwareMap) = (elit_initialized);
        b1 := b1 AND ((state0.dvar_M_HardwareMap_out_a_x2testing) <> (alg_a_x2testing(state0)));
        IF b1 THEN
            progress := TRUE;
            state1 := state0;

            state1.dvar_M_HardwareMap_out_a_x2testing := alg_a_x2testing(state0);

            state0 := state1;
        END_IF;
    END_IF;

    // Event "tau".
    IF NOT progress THEN
        b1 := (state0.dvar_M_HardwareMap) = (elit_initialized);
        b1 := b1 AND ((state0.dvar_M_HardwareMap_out_a_zdown) <> (alg_a_zdown(state0)));
        IF b1 THEN
            progress := TRUE;
            state1 := state0;

            state1.dvar_M_HardwareMap_out_a_zdown := alg_a_zdown(state0);

            state0 := state1;
        END_IF;
    END_IF;

    // Event "tau".
    IF NOT progress THEN
        b1 := (state0.dvar_M_HardwareMap) = (elit_initialized);
        b1 := b1 AND ((state0.dvar_M_HardwareMap_out_a_gripperclose) <> (alg_a_gripperclose(state0)));
        IF b1 THEN
            progress := TRUE;
            state1 := state0;

            state1.dvar_M_HardwareMap_out_a_gripperclose := alg_a_gripperclose(state0);

            state0 := state1;
        END_IF;
    END_IF;

    // Event "tau".
    IF NOT progress THEN
        b1 := (state0.dvar_M_HardwareMap) = (elit_initialized);
        b1 := b1 AND ((state0.dvar_M_HardwareMap_out_a_transfer2pickpos) <> (alg_a_transfer2pickpos(state0)));
        IF b1 THEN
            progress := TRUE;
            state1 := state0;

            state1.dvar_M_HardwareMap_out_a_transfer2pickpos := alg_a_transfer2pickpos(state0);

            state0 := state1;
        END_IF;
    END_IF;

    // Event "tau".
    IF NOT progress THEN
        b1 := (state0.dvar_M_HardwareMap) = (elit_initialized);
        b1 := b1 AND ((state0.dvar_M_HardwareMap_out_a_transfer2droppos) <> (alg_a_transfer2droppos(state0)));
        IF b1 THEN
            progress := TRUE;
            state1 := state0;

            state1.dvar_M_HardwareMap_out_a_transfer2droppos := alg_a_transfer2droppos(state0);

            state0 := state1;
        END_IF;
    END_IF;

    // Event "tau".
    IF NOT progress THEN
        b1 := (state0.dvar_M_HardwareMap) = (elit_initialized);
        b1 := b1 AND ((state0.dvar_M_HardwareMap_out_a_vacuum) <> (alg_a_vacuum(state0)));
        IF b1 THEN
            progress := TRUE;
            state1 := state0;

            state1.dvar_M_HardwareMap_out_a_vacuum := alg_a_vacuum(state0);

            state0 := state1;
        END_IF;
    END_IF;

    // Event "tau".
    IF NOT progress THEN
        b1 := (state0.dvar_M_HardwareMap) = (elit_initialized);
        b1 := b1 AND ((state0.dvar_M_HardwareMap_out_a_ejectpulse) <> (alg_a_ejectpulse(state0)));
        IF b1 THEN
            progress := TRUE;
            state1 := state0;

            state1.dvar_M_HardwareMap_out_a_ejectpulse := alg_a_ejectpulse(state0);

            state0 := state1;
        END_IF;
    END_IF;

    // Event "tau".
    IF NOT progress THEN
        b1 := (state0.dvar_M_HardwareMap) = (elit_initialized);
        b1 := b1 AND ((state0.dvar_M_HardwareMap_out_a_handlingready) <> (FALSE));
        IF b1 THEN
            progress := TRUE;
            state1 := state0;

            state1.dvar_M_HardwareMap_out_a_handlingready := FALSE;

            state0 := state1;
        END_IF;
    END_IF;

    // Event "tau".
    IF NOT progress THEN
        b1 := (state0.dvar_M_inventory1) = (elit_init2);
        b1 := b1 AND (alg_s_Dinitialized(state0));
        IF b1 THEN
            progress := TRUE;
            state1 := state0;

            state1.dvar_M_inventory1 := elit_wait_start;

            state0 := state1;
        END_IF;
    END_IF;

    // Event "tau".
    IF NOT progress THEN
        b1 := (state0.dvar_M_inventory1) = (elit_wait_start);
        b1 := b1 AND (ivar_s_Dstartbutton);
        IF b1 THEN
            progress := TRUE;
            state1 := state0;

            state1.dvar_M_inventory1 := elit_starting;

            state0 := state1;
        END_IF;
    END_IF;

    // Event "tau".
    IF NOT progress THEN
        b1 := (state0.dvar_M_inventory1) = (elit_starting);
        b1 := b1 AND (ivar_s_pusher1_in);
        b1 := b1 AND (NOT(ivar_s_product1));
        IF b1 THEN
            progress := TRUE;
            state1 := state0;

            state1.dvar_M_inventory1_a_pusher1 := TRUE;
            state1.dvar_M_inventory1 := elit_going;

            state0 := state1;
        END_IF;
    END_IF;

    // Event "tau".
    IF NOT progress THEN
        b1 := (state0.dvar_M_inventory1) = (elit_going);
        b1 := b1 AND (ivar_s_pusher1_out);
        b1 := b1 AND (ivar_s_stack1filled);
        IF b1 THEN
            progress := TRUE;
            state1 := state0;

            state1.dvar_M_inventory1_a_pusher1 := FALSE;
            state1.dvar_M_inventory1 := elit_starting;

            state0 := state1;
        END_IF;
    END_IF;

    // Event "tau".
    IF NOT progress THEN
        b1 := (state0.dvar_M_inventory2) = (elit_init2);
        b1 := b1 AND (alg_s_Dinitialized(state0));
        IF b1 THEN
            progress := TRUE;
            state1 := state0;

            state1.dvar_M_inventory2 := elit_wait_start;

            state0 := state1;
        END_IF;
    END_IF;

    // Event "tau".
    IF NOT progress THEN
        b1 := (state0.dvar_M_inventory2) = (elit_wait_start);
        b1 := b1 AND (ivar_s_Dstartbutton);
        IF b1 THEN
            progress := TRUE;
            state1 := state0;

            state1.dvar_M_inventory2 := elit_starting;

            state0 := state1;
        END_IF;
    END_IF;

    // Event "tau".
    IF NOT progress THEN
        b1 := (state0.dvar_M_inventory2) = (elit_starting);
        b1 := b1 AND (ivar_s_pusher2_in);
        b1 := b1 AND (NOT(ivar_s_product2));
        IF b1 THEN
            progress := TRUE;
            state1 := state0;

            state1.dvar_M_inventory2_a_pusher2 := TRUE;
            state1.dvar_M_inventory2 := elit_going;

            state0 := state1;
        END_IF;
    END_IF;

    // Event "tau".
    IF NOT progress THEN
        b1 := (state0.dvar_M_inventory2) = (elit_going);
        b1 := b1 AND (ivar_s_pusher2_out);
        b1 := b1 AND (ivar_s_stack2filled);
        IF b1 THEN
            progress := TRUE;
            state1 := state0;

            state1.dvar_M_inventory2_a_pusher2 := FALSE;
            state1.dvar_M_inventory2 := elit_starting;

            state0 := state1;
        END_IF;
    END_IF;

    // Event "tau".
    IF NOT progress THEN
        b1 := (state0.dvar_M_inventory3) = (elit_init2);
        b1 := b1 AND (alg_s_Dinitialized(state0));
        IF b1 THEN
            progress := TRUE;
            state1 := state0;

            state1.dvar_M_inventory3 := elit_wait_start;

            state0 := state1;
        END_IF;
    END_IF;

    // Event "tau".
    IF NOT progress THEN
        b1 := (state0.dvar_M_inventory3) = (elit_wait_start);
        b1 := b1 AND (ivar_s_Dstartbutton);
        IF b1 THEN
            progress := TRUE;
            state1 := state0;

            state1.dvar_M_inventory3 := elit_starting;

            state0 := state1;
        END_IF;
    END_IF;

    // Event "tau".
    IF NOT progress THEN
        b1 := (state0.dvar_M_inventory3) = (elit_starting);
        b1 := b1 AND (ivar_s_pusher3_in);
        b1 := b1 AND (NOT(ivar_s_product3));
        IF b1 THEN
            progress := TRUE;
            state1 := state0;

            state1.dvar_M_inventory3_a_pusher3 := TRUE;
            state1.dvar_M_inventory3 := elit_going;

            state0 := state1;
        END_IF;
    END_IF;

    // Event "tau".
    IF NOT progress THEN
        b1 := (state0.dvar_M_inventory3) = (elit_going);
        b1 := b1 AND (ivar_s_pusher3_out);
        b1 := b1 AND (ivar_s_stack3filled);
        IF b1 THEN
            progress := TRUE;
            state1 := state0;

            state1.dvar_M_inventory3_a_pusher3 := FALSE;
            state1.dvar_M_inventory3 := elit_starting;

            state0 := state1;
        END_IF;
    END_IF;

    // Event "tau".
    IF NOT progress THEN
        b1 := (state0.dvar_M_vacuum) = (elit_init2);
        b1 := b1 AND (alg_s_Dinitialized(state0));
        IF b1 THEN
            progress := TRUE;
            state1 := state0;

            state1.dvar_M_vacuum := elit_wait_start;

            state0 := state1;
        END_IF;
    END_IF;

    // Event "tau".
    IF NOT progress THEN
        b1 := (state0.dvar_M_vacuum) = (elit_wait_start);
        b1 := b1 AND (ivar_s_Dstartbutton);
        IF b1 THEN
            progress := TRUE;
            state1 := state0;

            state1.dvar_M_vacuum := elit_starting;

            state0 := state1;
        END_IF;
    END_IF;

    // Event "tau".
    IF NOT progress THEN
        b1 := (state0.dvar_M_vacuum) = (elit_starting);
        b1 := b1 AND (ivar_s_product4);
        b1 := b1 AND (ivar_s_zpos_atup);
        b1 := b1 AND (NOT(ivar_s_vacuum));
        IF b1 THEN
            progress := TRUE;
            state1 := state0;

            state1.dvar_M_vacuum_a_transfer2pickpos := TRUE;
            state1.dvar_M_vacuum := elit_pickupvac;

            state0 := state1;
        END_IF;
    END_IF;

    // Event "tau".
    IF NOT progress THEN
        b1 := (state0.dvar_M_vacuum) = (elit_starting);
        b1 := b1 AND (ivar_s_vacuum);
        IF b1 THEN
            progress := TRUE;
            state1 := state0;

            state1.dvar_M_vacuum_a_transfer2droppos := TRUE;
            state1.dvar_M_vacuum := elit_pickupvac;

            state0 := state1;
        END_IF;
    END_IF;

    // Event "tau".
    IF NOT progress THEN
        b1 := (state0.dvar_M_vacuum) = (elit_pickupvac);
        b1 := b1 AND (ivar_s_transfer_atpickup);
        b1 := b1 AND (NOT(ivar_s_vacuum));
        IF b1 THEN
            progress := TRUE;
            state1 := state0;

            state1.dvar_M_vacuum_a_transfer2pickpos := FALSE;
            state1.dvar_M_vacuum_a_vacuum := TRUE;
            state1.dvar_M_vacuum := elit_testingdrop;

            state0 := state1;
        END_IF;
    END_IF;

    // Event "tau".
    IF NOT progress THEN
        b1 := (state0.dvar_M_vacuum) = (elit_pickupvac);
        b1 := b1 AND (ivar_s_transfer_atdrop);
        IF b1 THEN
            progress := TRUE;
            state1 := state0;

            state1.dvar_M_vacuum_a_vacuum := FALSE;
            state1.dvar_M_vacuum_a_ejectpulse := TRUE;
            state1.dvar_M_vacuum_a_transfer2pickpos := TRUE;
            state1.dvar_M_vacuum_a_transfer2droppos := FALSE;
            state1.dvar_M_vacuum := elit_rest;

            state0 := state1;
        END_IF;
    END_IF;

    // Event "tau".
    IF NOT progress THEN
        b1 := (state0.dvar_M_vacuum) = (elit_testingdrop);
        b1 := b1 AND (ivar_s_vacuum);
        IF b1 THEN
            progress := TRUE;
            state1 := state0;

            state1.dvar_M_vacuum_a_transfer2droppos := TRUE;
            state1.dvar_M_vacuum := elit_starting;

            state0 := state1;
        END_IF;
    END_IF;

    // Event "tau".
    IF NOT progress THEN
        b1 := (state0.dvar_M_vacuum) = (elit_rest);
        b1 := b1 AND (ivar_s_transfer_athalfway);
        IF b1 THEN
            progress := TRUE;
            state1 := state0;

            state1.dvar_M_vacuum_a_transfer2pickpos := FALSE;
            state1.dvar_M_vacuum_a_transfer2droppos := FALSE;
            state1.dvar_M_vacuum_a_vacuum := FALSE;
            state1.dvar_M_vacuum_a_ejectpulse := FALSE;
            state1.dvar_M_vacuum := elit_starting;

            state0 := state1;
        END_IF;
    END_IF;

    // Done with events?
    IF NOT progress THEN
        EXIT;
    END_IF;

    // Protect against events that are always enabled.
    loopCount := loopCount + 1;
    IF loopCount >= 100 THEN
        loopsKilled := loopsKilled + 1;
        EXIT;
    END_IF;
END_WHILE;

END_PROGRAM

// ---- CIF/derivcvar_M_HardwareMap_t.TcPOU
FUNCTION derivcvar_M_HardwareMap_t : LREAL
VAR_INPUT
	state: STATE;
END_VAR

derivcvar_M_HardwareMap_t := 1.0;

END_FUNCTION

// ---- CIF/alg_s_Dinitialized.TcPOU
FUNCTION alg_s_Dinitialized : BOOL
VAR_INPUT
	state: STATE;
END_VAR

alg_s_Dinitialized := (state.dvar_M_HardwareMap) = (elit_initialized);

END_FUNCTION

// ---- CIF/projArray0.TcPOU
FUNCTION projArray0 : BOOL
VAR_INPUT
	arr: ARRAY[0..2] OF BOOL;
	idx: DINT;
END_VAR

projArray0 := arr[normProjIdx(idx, 3)];

END_FUNCTION

// ---- CIF/normProjIdx.TcPOU
FUNCTION normProjIdx : DINT
VAR_INPUT
	idx: DINT;
	size: DINT;
END_VAR
VAR
	tmp: DINT;
END_VAR

tmp := idx;
IF tmp < 0 THEN
    tmp := size + tmp;
END_IF;
normProjIdx := tmp;

END_FUNCTION

// ---- CIF/makeArray0.TcPOU
FUNCTION makeArray0 : ARRAY[0..2] OF BOOL
VAR_INPUT
	elem0: BOOL;
	elem1: BOOL;
	elem2: BOOL;
END_VAR
VAR
	rslt: ARRAY[0..2] OF BOOL;
END_VAR

rslt[0] := elem0;
rslt[1] := elem1;
rslt[2] := elem2;
makeArray0 := rslt;

END_FUNCTION

// ---- CIF/alg_a_Dstartled.TcPOU
FUNCTION alg_a_Dstartled : BOOL
VAR_INPUT
	state: STATE;
END_VAR

alg_a_Dstartled := alg_M_example_controller_a_Dstartled(state);

END_FUNCTION

// ---- CIF/alg_M_example_controller_a_Dstartled.TcPOU
FUNCTION alg_M_example_controller_a_Dstartled : BOOL
VAR_INPUT
	state: STATE;
END_VAR

alg_M_example_controller_a_Dstartled := (state.dvar_M_example_controller) = (elit_running);

END_FUNCTION

// ---- CIF/alg_a_pusher1.TcPOU
FUNCTION alg_a_pusher1 : BOOL
VAR_INPUT
	state: STATE;
END_VAR

alg_a_pusher1 := FALSE;

END_FUNCTION

// ---- CIF/alg_a_pusher2.TcPOU
FUNCTION alg_a_pusher2 : BOOL
VAR_INPUT
	state: STATE;
END_VAR

alg_a_pusher2 := FALSE;

END_FUNCTION

// ---- CIF/alg_a_pusher3.TcPOU
FUNCTION alg_a_pusher3 : BOOL
VAR_INPUT
	state: STATE;
END_VAR

alg_a_pusher3 := FALSE;

END_FUNCTION

// ---- CIF/alg_a_x2distributing.TcPOU
FUNCTION alg_a_x2distributing : BOOL
VAR_INPUT
	state: STATE;
END_VAR

alg_a_x2distributing := state.dvar_M_example_controller_a_x2distributing;

END_FUNCTION

// ---- CIF/alg_a_x2testing.TcPOU
FUNCTION alg_a_x2testing : BOOL
VAR_INPUT
	state: STATE;
END_VAR

alg_a_x2testing := FALSE;

END_FUNCTION

// ---- CIF/alg_a_zdown.TcPOU
FUNCTION alg_a_zdown : BOOL
VAR_INPUT
	state: STATE;
END_VAR

alg_a_zdown := state.dvar_M_example_controller_a_zdown;

END_FUNCTION

// ---- CIF/alg_a_gripperclose.TcPOU
FUNCTION alg_a_gripperclose : BOOL
VAR_INPUT
	state: STATE;
END_VAR

alg_a_gripperclose := FALSE;

END_FUNCTION

// ---- CIF/alg_a_transfer2pickpos.TcPOU
FUNCTION alg_a_transfer2pickpos : BOOL
VAR_INPUT
	state: STATE;
END_VAR

alg_a_transfer2pickpos := FALSE;

END_FUNCTION

// ---- CIF/alg_a_transfer2droppos.TcPOU
FUNCTION alg_a_transfer2droppos : BOOL
VAR_INPUT
	state: STATE;
END_VAR

alg_a_transfer2droppos := FALSE;

END_FUNCTION

// ---- CIF/alg_a_vacuum.TcPOU
FUNCTION alg_a_vacuum : BOOL
VAR_INPUT
	state: STATE;
END_VAR

alg_a_vacuum := FALSE;

END_FUNCTION

// ---- CIF/alg_a_ejectpulse.TcPOU
FUNCTION alg_a_ejectpulse : BOOL
VAR_INPUT
	state: STATE;
END_VAR

alg_a_ejectpulse := FALSE;

END_FUNCTION

// ---- UNITY/UNITY.TcPOU
PROGRAM UNITY
VAR
END_VAR

// Mapping program - DO NOT CHANGE

//// \\\\ DISTRIBUTING //// \\\\

/// ACTUATORS
// a_pusher1
GVLs.Actuator[0].oToggle 	:= MAIN.state0.dvar_M_HardwareMap_out_a_pusher1;
// a_pusher2
GVLs.Actuator[1].oToggle 	:= MAIN.state0.dvar_M_HardwareMap_out_a_pusher2;
// a_pusher3
GVLs.Actuator[2].oToggle 	:= MAIN.state0.dvar_M_HardwareMap_out_a_pusher3;

/// SENSORS
// s_pusher1_in
INPUTS.ivar_s_pusher1_in 	:= GVLs.INDICATORLIGHT[0].iActive;
// s_pusher1_out
INPUTS.ivar_s_pusher1_out 	:= GVLs.INDICATORLIGHT[1].iActive;
// s_stack1filled
INPUTS.ivar_s_stack1filled 	:= GVLs.INDICATORLIGHT[2].iActive;
// s_product1
INPUTS.ivar_s_product1 		:= GVLs.INDICATORLIGHT[3].iActive;
// s_pusher2_in
INPUTS.ivar_s_pusher2_in 	:= GVLs.INDICATORLIGHT[4].iActive;
// s_pusher2_out
INPUTS.ivar_s_pusher2_out 	:= GVLs.INDICATORLIGHT[5].iActive;
// s_stack2filled
INPUTS.ivar_s_stack2filled 	:= GVLs.INDICATORLIGHT[6].iActive;
// s_product2
INPUTS.ivar_s_product2 		:= GVLs.INDICATORLIGHT[7].iActive;
// s_pusher3_in
INPUTS.ivar_s_pusher3_in 	:= GVLs.INDICATORLIGHT[8].iActive;
// s_pusher3_out
INPUTS.ivar_s_pusher3_out 	:= GVLs.INDICATORLIGHT[9].iActive;
// s_stack3filled
INPUTS.ivar_s_stack3filled 	:= GVLs.INDICATORLIGHT[10].iActive;
// s_product3
INPUTS.ivar_s_product3 		:= GVLs.INDICATORLIGHT[11].iActive;
// s_handlingbusy
INPUTS.ivar_s_handlingbusy 	:= GVLs.INDICATORLIGHT[12].iActive;

/// CONTROL PANEL
// s_Dstartbutton
INPUTS.ivar_s_Dstartbutton	:= GVLs.INDICATORLIGHT[13].iActive;
// s_Dstopbutton
INPUTS.ivar_s_Dstopbutton	:= NOT GVLs.INDICATORLIGHT[14].iActive;
// s_Dautoswitch
INPUTS.ivar_s_Dautoswitch	:= GVLs.INDICATORLIGHT[15].iActive;
// s_Dresetbutton
INPUTS.ivar_s_Dresetbutton	:= GVLs.INDICATORLIGHT[16].iActive;
// s_Din4
INPUTS.ivar_s_Din4			:= GVLs.INDICATORLIGHT[17].iActive;
// s_Din5
INPUTS.ivar_s_Din5			:= GVLs.INDICATORLIGHT[18].iActive;
// s_Din6
INPUTS.ivar_s_Din6			:= GVLs.INDICATORLIGHT[19].iActive;
// s_Din7
INPUTS.ivar_s_Din7			:= GVLs.INDICATORLIGHT[20].iActive;
// a_Dstartled
GVLS.INDICATORLIGHT[21].oActive	:= MAIN.state0.dvar_M_HardwareMap_out_a_Dstartled;
// a_Dresetled
GVLS.INDICATORLIGHT[22].oActive	:= MAIN.state0.dvar_M_HardwareMap_out_a_Dresetled;
// a_DledQ1
GVLS.INDICATORLIGHT[23].oActive	:= MAIN.state0.dvar_M_HardwareMap_out_a_DledQ1;
// a_DledQ2
GVLS.INDICATORLIGHT[24].oActive	:= MAIN.state0.dvar_M_HardwareMap_out_a_DledQ2;
// a_Dout4
GVLS.INDICATORLIGHT[25].oActive	:= MAIN.state0.dvar_M_HardwareMap_out_a_Dout4;
// a_Dout5
GVLS.INDICATORLIGHT[26].oActive	:= MAIN.state0.dvar_M_HardwareMap_out_a_Dout5;
// a_Dout6
GVLS.INDICATORLIGHT[27].oActive	:= MAIN.state0.dvar_M_HardwareMap_out_a_Dout6;
// a_Dout7
GVLS.INDICATORLIGHT[28].oActive	:= MAIN.state0.dvar_M_HardwareMap_out_a_Dout7;

//// \\\\ HANDLING \\\\ ////

/// ACTUATORS
// a_x2distributing
GVLs.Actuator[3].oToggle 	:= MAIN.state0.dvar_M_HardwareMap_out_a_x2distributing;
// a_x2testing
GVLs.Actuator[4].oToggle 	:= MAIN.state0.dvar_M_HardwareMap_out_a_x2testing;
// a_zdown
GVLs.Actuator[5].oToggle 	:= MAIN.state0.dvar_M_HardwareMap_out_a_zdown;
// a_gripperclose
GVLs.Actuator[6].oToggle 	:= MAIN.state0.dvar_M_HardwareMap_out_a_gripperclose;
// a_transfer2pickpos
GVLs.Actuator[7].oToggle 	:= MAIN.state0.dvar_M_HardwareMap_out_a_transfer2pickpos;
// transfer2droppos
GVLs.Actuator[8].oToggle 	:= MAIN.state0.dvar_M_HardwareMap_out_a_transfer2droppos;
// a_vacuum
GVLs.Actuator[9].oToggle 	:= MAIN.state0.dvar_M_HardwareMap_out_a_vacuum;
// a_ejectpulse
GVLs.Actuator[10].oToggle	:= MAIN.state0.dvar_M_HardwareMap_out_a_ejectpulse;
// a_handlingready
GVLs.Actuator[11].oToggle 	:= MAIN.state0.dvar_M_HardwareMap_out_a_handlingready;

/// SENSORS
// s_xpos_at1
INPUTS.ivar_s_xpos_at1 				:= GVLs.INDICATORLIGHT[29].iActive;
// s_xpos_at2
INPUTS.ivar_s_xpos_at2 				:= GVLs.INDICATORLIGHT[30].iActive;
// s_xpos_at3
INPUTS.ivar_s_xpos_at3 				:= GVLs.INDICATORLIGHT[31].iActive;
// s_xpos_atdrop
INPUTS.ivar_s_xpos_atdrop 			:= GVLs.INDICATORLIGHT[32].iActive;
// s_zpos_atup
INPUTS.ivar_s_zpos_atup				:= GVLs.INDICATORLIGHT[33].iActive;
// s_zpos_atdown
INPUTS.ivar_s_zpos_atdown			:= GVLs.INDICATORLIGHT[34].iActive;
// s_gripper
INPUTS.ivar_s_gripper 				:= GVLs.INDICATORLIGHT[35].iActive;
// s_transfer_atpickup
INPUTS.ivar_s_transfer_atpickup 	:= GVLs.INDICATORLIGHT[36].iActive;
// s_transfer_atdrop
INPUTS.ivar_s_transfer_atdrop 		:= GVLs.INDICATORLIGHT[37].iActive;
// s_transfer_athalfway
INPUTS.ivar_s_transfer_athalfway 	:= GVLs.INDICATORLIGHT[38].iActive;
// s_vacuum
INPUTS.ivar_s_vacuum 				:= GVLs.INDICATORLIGHT[39].iActive;
// s_product4
INPUTS.ivar_s_product4 				:= GVLs.INDICATORLIGHT[40].iActive;
// s_testingbusy
INPUTS.ivar_s_testingbusy 			:= GVLs.INDICATORLIGHT[41].iActive;

/// CONTROL PANEL
// s_Hstartbutton
INPUTS.ivar_s_Hstartbutton	:= GVLs.INDICATORLIGHT[42].iActive;
// s_Hstopbutton
INPUTS.ivar_s_Hstopbutton	:= NOT GVLs.INDICATORLIGHT[43].iActive;
// s_Hautoswitch
INPUTS.ivar_s_Hautoswitch	:= GVLs.INDICATORLIGHT[44].iActive;
// s_Hresetbutton
INPUTS.ivar_s_Hresetbutton	:= GVLs.INDICATORLIGHT[45].iActive;
// s_Hin4
INPUTS.ivar_s_Hin4			:= GVLs.INDICATORLIGHT[46].iActive;
// s_Hin5
INPUTS.ivar_s_Hin5			:= GVLs.INDICATORLIGHT[47].iActive;
// s_Hin6
INPUTS.ivar_s_Hin6			:= GVLs.INDICATORLIGHT[48].iActive;
// s_Hin7
INPUTS.ivar_s_Hin7			:= GVLs.INDICATORLIGHT[49].iActive;
// a_Hstartled
GVLS.INDICATORLIGHT[50].oActive	:= MAIN.state0.dvar_M_HardwareMap_out_a_Hstartled;
// a_Hresetled
GVLS.INDICATORLIGHT[51].oActive	:= MAIN.state0.dvar_M_HardwareMap_out_a_Hresetled;
// a_HledQ1
GVLS.INDICATORLIGHT[52].oActive	:= MAIN.state0.dvar_M_HardwareMap_out_a_HledQ1;
// a_HledQ2
GVLS.INDICATORLIGHT[53].oActive	:= MAIN.state0.dvar_M_HardwareMap_out_a_HledQ2;
// a_Hout4
GVLS.INDICATORLIGHT[54].oActive	:= MAIN.state0.dvar_M_HardwareMap_out_a_Hout4;
// a_Hout5
GVLS.INDICATORLIGHT[55].oActive	:= MAIN.state0.dvar_M_HardwareMap_out_a_Hout5;
// a_Hout6
GVLS.INDICATORLIGHT[56].oActive	:= MAIN.state0.dvar_M_HardwareMap_out_a_Hout6;
// a_Hout7
GVLS.INDICATORLIGHT[57].oActive	:= MAIN.state0.dvar_M_HardwareMap_out_a_Hout7;

END_PROGRAM

// ---- CIF/alg_a_DledQ1.TcPOU
FUNCTION alg_a_DledQ1 : BOOL
VAR_INPUT
	state: STATE;
END_VAR

alg_a_DledQ1 := FALSE;

END_FUNCTION

// ---- CIF/alg_a_DledQ2.TcPOU
FUNCTION alg_a_DledQ2 : BOOL
VAR_INPUT
	state: STATE;
END_VAR

alg_a_DledQ2 := FALSE;

END_FUNCTION

// ---- CIF/alg_a_Dresetled.TcPOU
FUNCTION alg_a_Dresetled : BOOL
VAR_INPUT
	state: STATE;
END_VAR

alg_a_Dresetled := FALSE;

END_FUNCTION

// ---- CIF/alg_a_handlingready.TcPOU
FUNCTION alg_a_handlingready : BOOL
VAR_INPUT
	state: STATE;
END_VAR

alg_a_handlingready := FALSE;

END_FUNCTION

// ---- CIF/alg_a_HledQ1.TcPOU
FUNCTION alg_a_HledQ1 : BOOL
VAR_INPUT
	state: STATE;
END_VAR

alg_a_HledQ1 := FALSE;

END_FUNCTION

// ---- CIF/alg_a_HledQ2.TcPOU
FUNCTION alg_a_HledQ2 : BOOL
VAR_INPUT
	state: STATE;
END_VAR

alg_a_HledQ2 := FALSE;

END_FUNCTION

// ---- CIF/alg_a_Hresetled.TcPOU
FUNCTION alg_a_Hresetled : BOOL
VAR_INPUT
	state: STATE;
END_VAR

alg_a_Hresetled := FALSE;

END_FUNCTION

// ---- CIF/alg_a_Hstartled.TcPOU
FUNCTION alg_a_Hstartled : BOOL
VAR_INPUT
	state: STATE;
END_VAR

alg_a_Hstartled := FALSE;

END_FUNCTION

// ---- CIF/alg_M_example_controller_godown.TcPOU
FUNCTION alg_M_example_controller_godown : ARRAY[0..2] OF BOOL
VAR_INPUT
	state: STATE;
END_VAR

alg_M_example_controller_godown := makeArray0(ivar_s_xpos_at1, ivar_s_xpos_at2, ivar_s_xpos_at3);

END_FUNCTION

// ---- CIF/alg_s_Hinitialized.TcPOU
FUNCTION alg_s_Hinitialized : BOOL
VAR_INPUT
	state: STATE;
END_VAR

alg_s_Hinitialized := (state.dvar_M_HardwareMap) = (elit_initialized);

END_FUNCTION
